TYPE motor_info_datagrid :
STRUCT
	speed : LREAL;
	torque : LREAL;
	errortype : UDINT;
	errorid : UDINT;
END_STRUCT
END_TYPE

(* stored: Version 1.1.0.1, ProductVersion 3.1.4024.12
   DUT motor_info_datagrid: Id {3ba4319e-66c2-4f57-a3c8-f2a18bb2c71a} *)
